{attribute 'qualified_only'}
VAR_GLOBAL
	bOut1 	AT%Q*	: BOOL;
	bIn1 	AT%I*	: BOOL;	
END_VAR

(* stored: Version 1.1.0.1, ProductVersion 3.1.4024.10
   GVL IO: Id {a21286c5-545e-45f2-9901-9e6fb96fec56} *)
